(* PLC project motor_controller, Beckhoff Automation GmbH TwinCAT PLC Control 3.5.13.21 *)
(* stored: creationDateTime 2023-10-12T21:00:45.8485613, modificationDateTime 2023-10-12T21:00:45.8505595 *)

(* global variable list GVL *)
{attribute 'qualified_only'}
VAR_GLOBAL
	
// ***********************************************************************************
// Process inputs
// ***********************************************************************************

// WT ADD 
// Mode 
b_RED_Mode_Manual: BOOL; //Mode
b_RED_Mode_Laptop: BOOL; //Mode


// Temperature and Pressure Sensor
TemperatureAndPressure: STRING := 'TemperatureAndPressure';//***********************************************************
f_RED_Status_Temperature_Funnel_inlet : REAL; // [°C] 
f_RED_Status_Temperature_Funnel_outlet : REAL; // [°C] 
f_RED_Status_Temperature_Funnel_plate : REAL; // [°C] change to concrete pump temperature 

f_RED_Status_Pressure_Funnel_inlet : REAL; // [ bar]

f_RED_Status_Temperature_Concrete_Pump : REAL; // [°C] 
f_RED_Status_Pressure_Concrete_Pump: REAL; // [ bar]

END_VAR
